// TIA Portal V15.1 export
// export: Created 2026-01-15T16:29:47.6176807Z, ExportSetting WithDefaults, WithReadOnly, DisplayName Totally Integrated Automation Portal, DisplayVersion V15.1 Update 8, DisplayName TIA Portal Openness, DisplayVersion V15.1 Update 8, DisplayName STEP 7 Professional, DisplayVersion V15.1 Update 8, DisplayName WinCC Advanced, DisplayVersion V15.1 Update 8
FUNCTION "FCXL_CCD_AGG12345" : Void   // FC9, LAD
{ S7_Optimized_Access := 'TRUE' }
VERSION : 0.1
// stored: AutoNumber true, CodeModifiedDate 2026-01-15T16:25:54.9938096Z, CompileDate 2026-01-15T16:25:55.0442288Z, CreationDate 2026-01-15T16:24:02.4619467Z, HandleErrorsWithinBlock false, InterfaceModifiedDate 2024-08-08T03:04:52.4075121Z, IsConsistent true, IsIECCheckEnabled false, IsKnowHowProtected false, IsWriteProtected false, LibraryConformanceStatus Error: The block contains calls of single instances. Warning: The object contains access to global data blocks. Warning: The block contains direct access to inputs, outputs, bit memories, indirect access to the registry or indirect access to external memory areas that are unknown at the time of compilation., ModifiedDate 2026-01-15T16:25:54.9938096Z, ParameterModified 2024-08-08T03:04:52.4075121Z, PLCSimAdvancedSupport false, SetENOAutomatically False, StructureModified 2024-08-08T03:04:52.4075121Z, UDAEnableTagReadback false
   VAR_TEMP   // added for the SCL form of the ladder/FBD networks
      _w1 : Bool;
      _w2 : Bool;
      _w3 : Bool;
   END_VAR
BEGIN

REGION Network 1: XU LY CAN AGG1
   // Các chân PV_IN và chân WR_IN không có tác dụng cho FB6
   // Mục đích của FB6 là xử lý giá trị cân WE_AG1 để biến nó thành cân có thể cân nhiều thành phần,bằng cách trừ bì thành phần đã cân trước đó
   // Chú ý tránh nhầm lẫn:
   // WE_AG1 hay những biến có chữ AG1 chưa chắc là dành cho cân thành phần AGG1 nhé, có thể nó là đang nói đến cái cân (thường có chữ W ở trước, ví dụ WE_AG1 là cái cân AGG nhé)
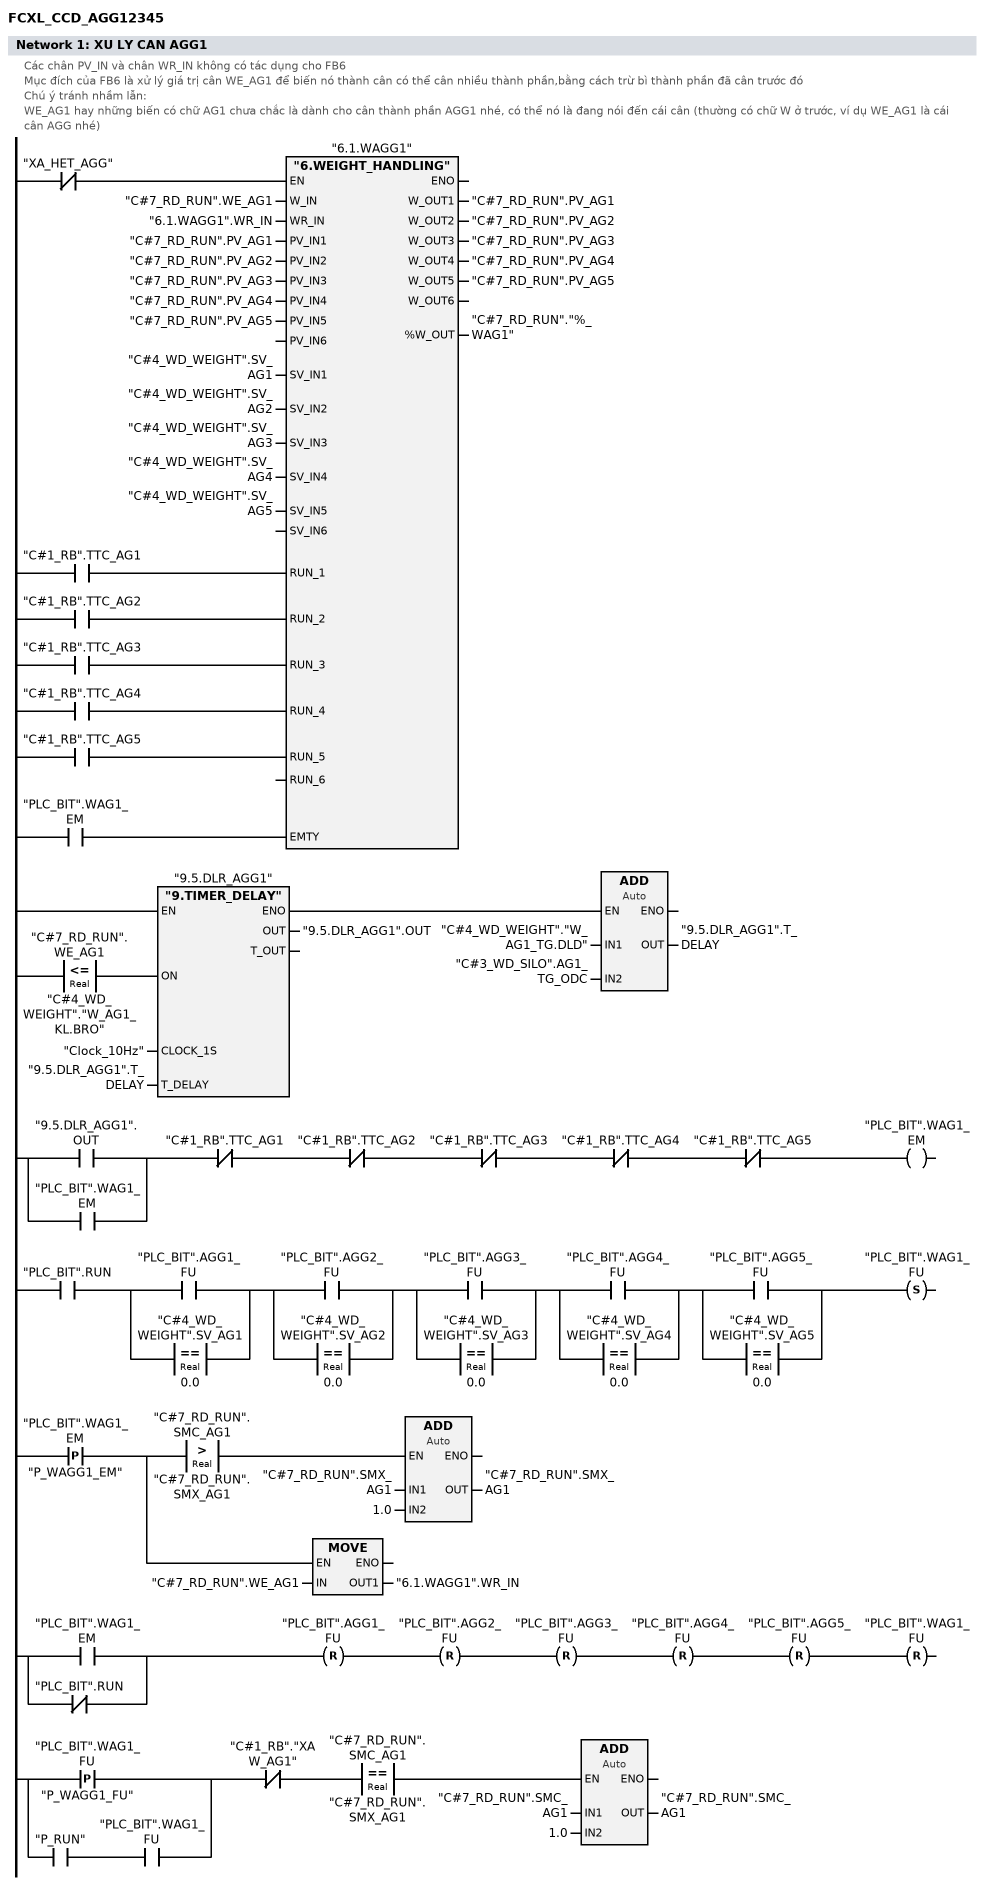
   RUNG wire#powerrail
      I_Contact( "XA_HET_AGG" )
      "6.1.WAGG1"(RUN_1 := wire#w1, RUN_2 := wire#w2, RUN_3 := wire#w3, RUN_4 := wire#w4, RUN_5 := wire#w5, EMTY := wire#w6, W_IN := "C#7_RD_RUN".WE_AG1, WR_IN := "6.1.WAGG1".WR_IN, PV_IN1 := "C#7_RD_RUN".PV_AG1, PV_IN2 := "C#7_RD_RUN".PV_AG2, PV_IN3 := "C#7_RD_RUN".PV_AG3, PV_IN4 := "C#7_RD_RUN".PV_AG4, PV_IN5 := "C#7_RD_RUN".PV_AG5, PV_IN6 :=, SV_IN1 := "C#4_WD_WEIGHT".SV_AG1, SV_IN2 := "C#4_WD_WEIGHT".SV_AG2, SV_IN3 := "C#4_WD_WEIGHT".SV_AG3, SV_IN4 := "C#4_WD_WEIGHT".SV_AG4, SV_IN5 := "C#4_WD_WEIGHT".SV_AG5, SV_IN6 :=, RUN_6 :=, W_OUT1 => "C#7_RD_RUN".PV_AG1, W_OUT2 => "C#7_RD_RUN".PV_AG2, W_OUT3 => "C#7_RD_RUN".PV_AG3, W_OUT4 => "C#7_RD_RUN".PV_AG4, W_OUT5 => "C#7_RD_RUN".PV_AG5, W_OUT6 =>, "%W_OUT" => "C#7_RD_RUN"."%_WAG1")
   END_RUNG
   RUNG wire#powerrail
      Contact( "C#1_RB".TTC_AG1 )
   END_RUNG wire#w1
   RUNG wire#powerrail
      Contact( "C#1_RB".TTC_AG2 )
   END_RUNG wire#w2
   RUNG wire#powerrail
      Contact( "C#1_RB".TTC_AG3 )
   END_RUNG wire#w3
   RUNG wire#powerrail
      Contact( "C#1_RB".TTC_AG4 )
   END_RUNG wire#w4
   RUNG wire#powerrail
      Contact( "C#1_RB".TTC_AG5 )
   END_RUNG wire#w5
   RUNG wire#powerrail
      Contact( "PLC_BIT".WAG1_EM )
   END_RUNG wire#w6
   RUNG wire#powerrail
      "9.5.DLR_AGG1"(ON := wire#w7, CLOCK_1S := "Clock_10Hz", T_DELAY := "9.5.DLR_AGG1".T_DELAY, OUT => "9.5.DLR_AGG1".OUT, T_OUT =>)
      Add(in1 := "C#4_WD_WEIGHT"."W_AG1_TG.DLD", in2 := "C#3_WD_SILO".AG1_TG_ODC, out => "9.5.DLR_AGG1".T_DELAY)
   END_RUNG
   RUNG wire#powerrail
      { S7_Templates := "SrcType := Real" } LE_Contact(in1 := "C#7_RD_RUN".WE_AG1, in2 := "C#4_WD_WEIGHT"."W_AG1_KL.BRO")
   END_RUNG wire#w7
   RUNG wire#powerrail
      Contact( "9.5.DLR_AGG1".OUT )
      wire#w8
      I_Contact( "C#1_RB".TTC_AG1 )
      I_Contact( "C#1_RB".TTC_AG2 )
      I_Contact( "C#1_RB".TTC_AG3 )
      I_Contact( "C#1_RB".TTC_AG4 )
      I_Contact( "C#1_RB".TTC_AG5 )
      Coil( "PLC_BIT".WAG1_EM )
   END_RUNG
   RUNG wire#powerrail
      Contact( "PLC_BIT".WAG1_EM )
   END_RUNG wire#w8
   RUNG wire#powerrail
      Contact( "PLC_BIT".RUN )
      wire#w9
      Contact( "PLC_BIT".AGG1_FU )
      wire#w10
      Contact( "PLC_BIT".AGG2_FU )
      wire#w11
      Contact( "PLC_BIT".AGG3_FU )
      wire#w12
      Contact( "PLC_BIT".AGG4_FU )
      wire#w13
      Contact( "PLC_BIT".AGG5_FU )
      wire#w14
      S_Coil( "PLC_BIT".WAG1_FU )
   END_RUNG
   RUNG wire#w9
      { S7_Templates := "SrcType := Real" } EQ_Contact(in1 := "C#4_WD_WEIGHT".SV_AG1, in2 := 0.0)
   END_RUNG wire#w10
   RUNG wire#w10
      { S7_Templates := "SrcType := Real" } EQ_Contact(in1 := "C#4_WD_WEIGHT".SV_AG2, in2 := 0.0)
   END_RUNG wire#w11
   RUNG wire#w11
      { S7_Templates := "SrcType := Real" } EQ_Contact(in1 := "C#4_WD_WEIGHT".SV_AG3, in2 := 0.0)
   END_RUNG wire#w12
   RUNG wire#w12
      { S7_Templates := "SrcType := Real" } EQ_Contact(in1 := "C#4_WD_WEIGHT".SV_AG4, in2 := 0.0)
   END_RUNG wire#w13
   RUNG wire#w13
      { S7_Templates := "SrcType := Real" } EQ_Contact(in1 := "C#4_WD_WEIGHT".SV_AG5, in2 := 0.0)
   END_RUNG wire#w14
   RUNG wire#powerrail
      P_Contact(operand := "PLC_BIT".WAG1_EM, bit := "P_WAGG1_EM")
      wire#w15
      { S7_Templates := "SrcType := Real" } GT_Contact(in1 := "C#7_RD_RUN".SMC_AG1, in2 := "C#7_RD_RUN".SMX_AG1)
      Add(in1 := "C#7_RD_RUN".SMX_AG1, in2 := 1.0, out => "C#7_RD_RUN".SMX_AG1)
   END_RUNG
   RUNG wire#w15
      Move(in := "C#7_RD_RUN".WE_AG1, out1 => "6.1.WAGG1".WR_IN)
   END_RUNG
   RUNG wire#powerrail
      Contact( "PLC_BIT".WAG1_EM )
      wire#w16
      R_Coil( "PLC_BIT".AGG1_FU )
      R_Coil( "PLC_BIT".AGG2_FU )
      R_Coil( "PLC_BIT".AGG3_FU )
      R_Coil( "PLC_BIT".AGG4_FU )
      R_Coil( "PLC_BIT".AGG5_FU )
      R_Coil( "PLC_BIT".WAG1_FU )
   END_RUNG
   RUNG wire#powerrail
      I_Contact( "PLC_BIT".RUN )
   END_RUNG wire#w16
   RUNG wire#powerrail
      P_Contact(operand := "PLC_BIT".WAG1_FU, bit := "P_WAGG1_FU")
      wire#w17
      I_Contact( "C#1_RB"."XA W_AG1" )
      { S7_Templates := "SrcType := Real" } EQ_Contact(in1 := "C#7_RD_RUN".SMC_AG1, in2 := "C#7_RD_RUN".SMX_AG1)
      Add(in1 := "C#7_RD_RUN".SMC_AG1, in2 := 1.0, out => "C#7_RD_RUN".SMC_AG1)
   END_RUNG
   RUNG wire#powerrail
      Contact( "P_RUN" )
      Contact( "PLC_BIT".WAG1_FU )
   END_RUNG wire#w17
   // the same network as SCL:
   IF NOT "XA_HET_AGG" THEN
       "6.1.WAGG1"(W_IN := "C#7_RD_RUN".WE_AG1,   // "6.WEIGHT_HANDLING"
                   WR_IN := "6.1.WAGG1".WR_IN,
                   PV_IN1 := "C#7_RD_RUN".PV_AG1,
                   PV_IN2 := "C#7_RD_RUN".PV_AG2,
                   PV_IN3 := "C#7_RD_RUN".PV_AG3,
                   PV_IN4 := "C#7_RD_RUN".PV_AG4,
                   PV_IN5 := "C#7_RD_RUN".PV_AG5,
                   SV_IN1 := "C#4_WD_WEIGHT".SV_AG1,
                   SV_IN2 := "C#4_WD_WEIGHT".SV_AG2,
                   SV_IN3 := "C#4_WD_WEIGHT".SV_AG3,
                   SV_IN4 := "C#4_WD_WEIGHT".SV_AG4,
                   SV_IN5 := "C#4_WD_WEIGHT".SV_AG5,
                   RUN_1 := "C#1_RB".TTC_AG1,
                   RUN_2 := "C#1_RB".TTC_AG2,
                   RUN_3 := "C#1_RB".TTC_AG3,
                   RUN_4 := "C#1_RB".TTC_AG4,
                   RUN_5 := "C#1_RB".TTC_AG5,
                   EMTY := "PLC_BIT".WAG1_EM,
                   W_OUT1 => "C#7_RD_RUN".PV_AG1,
                   W_OUT2 => "C#7_RD_RUN".PV_AG2,
                   W_OUT3 => "C#7_RD_RUN".PV_AG3,
                   W_OUT4 => "C#7_RD_RUN".PV_AG4,
                   W_OUT5 => "C#7_RD_RUN".PV_AG5,
                   "%W_OUT" => "C#7_RD_RUN"."%_WAG1");
   END_IF;
   "9.5.DLR_AGG1"(ON := "C#7_RD_RUN".WE_AG1 <= "C#4_WD_WEIGHT"."W_AG1_KL.BRO",   // "9.TIMER_DELAY"
                  CLOCK_1S := "Clock_10Hz",
                  T_DELAY := "9.5.DLR_AGG1".T_DELAY,
                  OUT => "9.5.DLR_AGG1".OUT,
                  ENO => #_w1);
   IF #_w1 THEN "9.5.DLR_AGG1".T_DELAY := "C#4_WD_WEIGHT"."W_AG1_TG.DLD" + "C#3_WD_SILO".AG1_TG_ODC; END_IF;
   "PLC_BIT".WAG1_EM := ("9.5.DLR_AGG1".OUT OR "PLC_BIT".WAG1_EM) AND NOT "C#1_RB".TTC_AG1 AND NOT "C#1_RB".TTC_AG2 AND NOT "C#1_RB".TTC_AG3 AND NOT "C#1_RB".TTC_AG4 AND NOT "C#1_RB".TTC_AG5;
   IF "PLC_BIT".RUN AND ("PLC_BIT".AGG1_FU OR ("C#4_WD_WEIGHT".SV_AG1 = 0.0)) AND ("PLC_BIT".AGG2_FU OR ("C#4_WD_WEIGHT".SV_AG2 = 0.0)) AND ("PLC_BIT".AGG3_FU OR ("C#4_WD_WEIGHT".SV_AG3 = 0.0)) AND ("PLC_BIT".AGG4_FU OR ("C#4_WD_WEIGHT".SV_AG4 = 0.0)) AND ("PLC_BIT".AGG5_FU OR ("C#4_WD_WEIGHT".SV_AG5 = 0.0)) THEN
       "PLC_BIT".WAG1_FU := TRUE;
   END_IF;
   #_w2 := "PLC_BIT".WAG1_EM AND NOT "P_WAGG1_EM";   // rising edge of "PLC_BIT".WAG1_EM
   "P_WAGG1_EM" := "PLC_BIT".WAG1_EM;
   IF #_w2 AND ("C#7_RD_RUN".SMC_AG1 > "C#7_RD_RUN".SMX_AG1) THEN
       "C#7_RD_RUN".SMX_AG1 := "C#7_RD_RUN".SMX_AG1 + 1.0;
   END_IF;
   IF #_w2 THEN "6.1.WAGG1".WR_IN := "C#7_RD_RUN".WE_AG1; END_IF;
   IF "PLC_BIT".WAG1_EM OR NOT "PLC_BIT".RUN THEN
       "PLC_BIT".AGG1_FU := FALSE;
       "PLC_BIT".AGG2_FU := FALSE;
       "PLC_BIT".AGG3_FU := FALSE;
       "PLC_BIT".AGG4_FU := FALSE;
       "PLC_BIT".AGG5_FU := FALSE;
       "PLC_BIT".WAG1_FU := FALSE;
   END_IF;
   #_w3 := "PLC_BIT".WAG1_FU AND NOT "P_WAGG1_FU";   // rising edge of "PLC_BIT".WAG1_FU
   "P_WAGG1_FU" := "PLC_BIT".WAG1_FU;
   IF (#_w3 OR ("P_RUN" AND "PLC_BIT".WAG1_FU)) AND NOT "C#1_RB"."XA W_AG1" AND ("C#7_RD_RUN".SMC_AG1 = "C#7_RD_RUN".SMX_AG1) THEN
       "C#7_RD_RUN".SMC_AG1 := "C#7_RD_RUN".SMC_AG1 + 1.0;
   END_IF;
END_REGION
END_FUNCTION
